TEXTLIST ProBox_Version
  Version = 'R1.13.0'
  Company = 'Swisslog/PTC'
   = ''
END_TEXTLIST

(* stored: Version 1.1.0.1, ProductVersion 3.1.4024.9
   TextList ProBox_Version: Id {55ce7c6f-e8ca-4a47-adca-dd570e8fe412} *)
